FUNCTION CompareAnyType : E_GeneralResult
VAR_INPUT
	A					: __SYSTEM.AnyType; // A and B have to be same type
	is					: E_Compare;
	B					: __SYSTEM.AnyType; // A and B have to be same type
END_VAR
VAR
END_VAR


CASE is OF
	E_Compare.EQUAL:
		CompareAnyType := IsEqualAnyType(A, B);
	E_Compare.NOT_EQUAL:
		CompareAnyType := IsNotEqualAnyType(A, B);
	E_Compare.LESS_THAN:
		CompareAnyType := IsLessThanAnyType(A, B);
	E_Compare.LOWER_THAN_OR_EQUAL:
		CompareAnyType := IsLessThanOrEqualAnyType(A, B);
	E_Compare.GREATER_THAN:
		CompareAnyType := IsGreaterThanAnyType(A, B);
	E_Compare.GREATER_THAN_OR_EQUAL:
		CompareAnyType := IsGreaterThanOrEqualAnyType(A, B);
END_CASE

END_FUNCTION

(* stored: Version 1.1.0.1, ProductVersion 3.1.4024.11
   POU CompareAnyType: Id {e0af17e2-781c-40ae-9369-407baf4161a9}, SpecialFunc None *)
